Fanuc KAREL source: ks00054.KL

-- PROVISIONAL review KL for V940-1; original PC SHA256 0f577b94fdd2f539563ddde6f04fa0834e544c93ab3430611ecdf3d60fa51b85
-- Incomplete behavior may be omitted. Consult companion uncertainty JSON. Do not deploy.
PROGRAM KS00054
%NOLOCKGROUP
BEGIN
  -- V9_ZERO_TABLE_METADATA_HINT layout=0001; no indexed target words; source/name/runtime held
  -- UNRESOLVED_PC offsets 5-13; opcodes 3F,75
  -- UNRESOLVED_PC offsets 18-27; opcodes 3F,75
  -- UNRESOLVED_PC offsets 32-45; opcodes 22,1D,23
  -- UNRESOLVED_PC offsets 50-54; opcodes 7F
END KS00054
